FUNCTION_BLOCK E_D_FF_ANY_HYS (* Data latch (d) flip flop with a Hysteresis *)
  (* Standard: 61499-1 Annex A; Description: Copyright (c) 2017 fortiss GmbH, HR Agrartechnik GmbH This program and the accompanying materials are made available under the terms of the Eclipse Public License 2.0 which is available at https://www.eclipse.org/legal/epl-2.0/ SPDX-License-Identifier: EPL-2.0 *)
  (* Version 1.0, 2026-04-17, Franz Höpfinger, HR Agrartechnik GmbH, E_D_FF copied and replace BOOL by ANY *)
  PACKAGE logiBUS::signalprocessing::hysteresis;
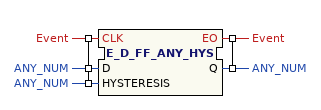
  EVENT_INPUT
    CLK WITH D, HYSTERESIS; (* Clock *)
  END_EVENT
  EVENT_OUTPUT
    EO WITH Q; (* Triggered if clock results in a change of Q *)
  END_EVENT
  VAR_INPUT
    D : ANY_NUM; (* Value to latch. Must be the same type as Q and HYSTERESIS *)
    HYSTERESIS : ANY_NUM; (* Hysteresis band. Must be the same type as D and Q *)
  END_VAR
  VAR_OUTPUT
    Q : ANY_NUM; (* Latched value. Must be the same type as D and HYSTERESIS *)
  END_VAR
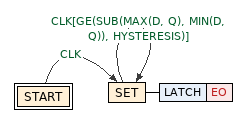
  EC_STATES
    START; (* Initial State *)
    SET : LATCH -> EO; (* Initialization *)
  END_STATES
  EC_TRANSITIONS
    SET TO SET := CLK[GE(SUB(MAX(D, Q), MIN(D, Q)), HYSTERESIS)];
    START TO SET := CLK;
  END_TRANSITIONS
  ALGORITHM LATCH IN ST: (* new algorithm *)
Q := D;
  END_ALGORITHM
END_FUNCTION_BLOCK
